KUKA KRL program: chk_w6_grp6_clo.src

&ACCESS RVO7
&COMMENT Check GRP AXOR Z6 CLOSE
DEF chk_w6_grp6_clo( )

; Check gripper axor CLOSE Z6.1/2/3/4
;//---- Start User-------

$TIMER[10] = 0
$TIMER_STOP[10] = FALSE

WAIT FOR (NOT $IN[509] and NOT $in[511] AND NOT $IN[513] AND NOT $IN[515])
WAIT FOR ($IN[510] and $in[512] AND $IN[514] AND $IN[516])

$TIMER_STOP[10] = TRUE
$TIMER[10] = 0

;//---- End User---------
END
